Universal Robots PolyScope program: test.urp

Program test (installation=custom_gripper_1 directory=/programs/usbdisk/new folder createdIn=5.14.5 lastSavedIn=5.14.5 robotSerialNumber=20225501312)
Calibrated DH parameters: a=[0.000177, -0.405867, -0.359302, -0.000009, 0.00008, 0]; d=[0.162556, -59.259033, 22.634856, 36.757695, 0.099775, 0.099535]; alpha=[1.570983, 0.00214, 0.004319, 1.570342, -1.569638, 0]; deltaTheta=[0, -0.302866, 6.171309, 0.414749, 0.000002, -0.000001]
InitVariablesNode
Robot Program (runOnlyOnce=false)
  Placeholder
